PROGRAM PRG_HEARTBEAT
VAR
	heartbeat AT %Q* : INT := 0;
	actuatorOn AT %Q* : BOOL;
END_VAR

heartbeat := heartbeat + 1;

IF heartbeat MOD 1000 = 0
	THEN actuatorOn := NOT actuatorOn;
END_IF

IF heartbeat MOD 30000 = 0
	THEN heartbeat := 0;
END_IF

END_PROGRAM

(* stored: Version 1.1.0.1, ProductVersion 3.1.4022.12
   POU PRG_HEARTBEAT: Id {07c2a92e-360a-4a8d-8ce4-0b8057ef0355}, SpecialFunc None *)
